Omron Sysmac Studio project TasimaBandi_Uygulamasi (Sysmac Studio 1.65.0.64007, StandardProject)

# Controller new_Controller_0: NX1P2-1040DT1 version 1.69
Task PrimaryTask (priority 4, period or condition 2000): Program0



PROGRAM Program0
VAR
    Start : BOOL;
    Band3 : TON;
    Band2 : TON;
    Band1 : BOOL;
    Stop : BOOL;
    Band_2 : BOOL;
    Band_3 : BOOL;
    Band_1 : BOOL;
    Start_Button : BOOL;
    Stop_Button : BOOL;
    TonStart : TON;
    TonStop : TON;
    AcilStop_Butonu : BOOL;
    Termik3_Ariza : BOOL;
    Bant3 : BOOL;
    Termik2_Ariza : BOOL;
    Bant2 : BOOL;
    Termik1_Ariza : BOOL;
    Bant1 : BOOL;
END_VAR
VAR
    _e1 : R_TRIG;
    _e2 : R_TRIG;
    _e3 : R_TRIG;
END_VAR

(* Section Section0: ladder, written here as Structured Text *)

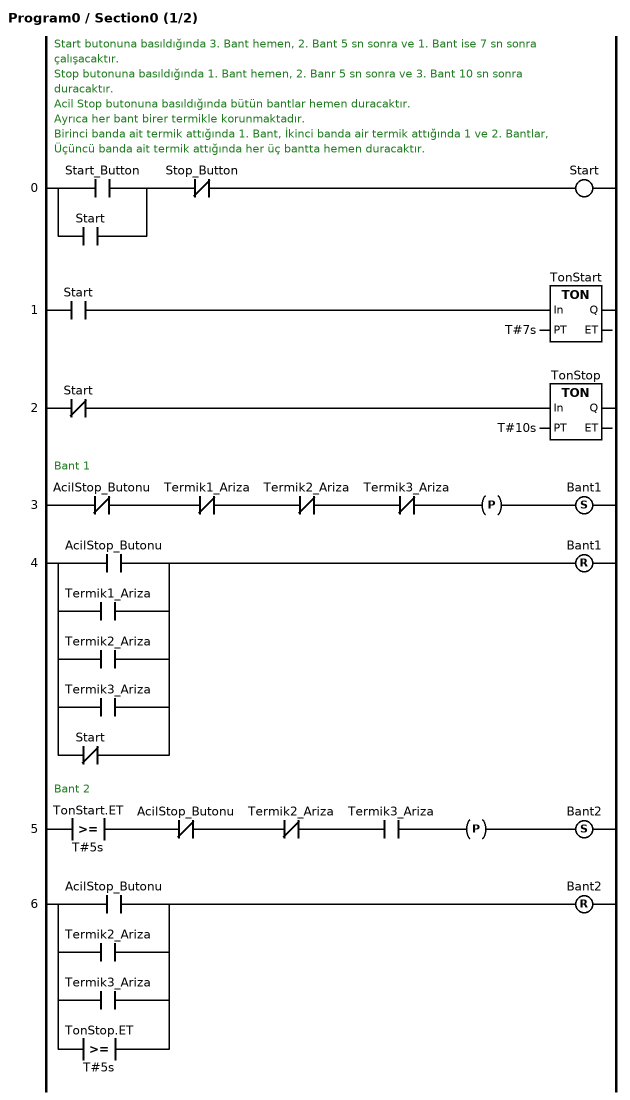
(* Rung 0: Start butonuna basıldığında 3. Bant hemen, 2. Bant 5 sn sonra ve 1. Bant ise 7 sn sonra çalışacaktır. / Stop butonuna basıldığında 1. Bant hemen, 2. Banr 5 sn sonra ve 3. Bant 10 sn sonra duracaktır. / Acil Stop butonuna basıldığında bütün bantlar hemen duracaktır. / Ayrıca her bant birer termikle korunmaktadır. / Birinci banda ait termik attığında 1. Bant, İkinci banda air termik attığında 1 ve 2. Bantlar, Üçüncü banda ait termik attığında her üç bantta hemen duracaktır. *)
Start := (Start_Button OR Start) AND NOT Stop_Button;
(* Rung 1 *)
TonStart(In := Start, PT := T#7s);
(* Rung 2 *)
TonStop(In := NOT Start, PT := T#10s);
(* Rung 3: Bant 1 *)
_e1(CLK := NOT AcilStop_Butonu AND NOT Termik1_Ariza AND NOT Termik2_Ariza AND NOT Termik3_Ariza);
IF _e1.Q THEN Bant1 := TRUE; END_IF;
(* Rung 4 *)
IF AcilStop_Butonu OR Termik1_Ariza OR Termik2_Ariza OR Termik3_Ariza OR NOT Start THEN
    Bant1 := FALSE;
END_IF;
(* Rung 5: Bant 2 *)
_e2(CLK := (TonStart.ET >= T#5s) AND NOT AcilStop_Butonu AND NOT Termik2_Ariza AND Termik3_Ariza);
IF _e2.Q THEN Bant2 := TRUE; END_IF;
(* Rung 6 *)
IF AcilStop_Butonu OR Termik2_Ariza OR Termik3_Ariza OR (TonStop.ET >= T#5s) THEN Bant2 := FALSE; END_IF;

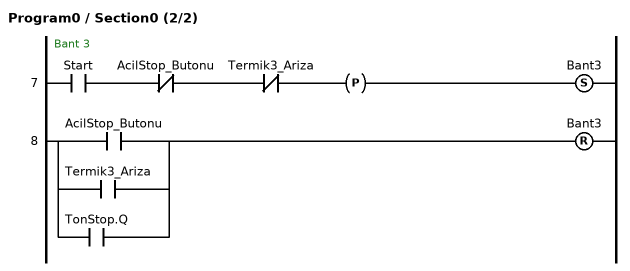
(* Rung 7: Bant 3 *)
_e3(CLK := Start AND NOT AcilStop_Butonu AND NOT Termik3_Ariza);
IF _e3.Q THEN Bant3 := TRUE; END_IF;
(* Rung 8 *)
IF AcilStop_Butonu OR Termik3_Ariza OR TonStop.Q THEN Bant3 := FALSE; END_IF;
END_PROGRAM